TYPE union_STATE_RS :
UNION
	byState		: BYTE;
	eState		: enum_FB_RS;
END_UNION
END_TYPE

(* stored: Version 1.1.0.1
   DUT union_STATE_RS: Id {8fb6fd03-2fad-449d-ac36-107455b6c3b8} *)
